FUNCTION_BLOCK RADIO_BOOL (* Radio Button BOOL Input *)
  (* Standard: 61499-1; Classification: HMI *)
  (* Version 0.3, 2004-06-21, JHC, Rockwell Automation, Updated documentation (REQ not inhibited). *)
  (* Version 0.2, 2004-06-08, JHC, Rockwell Automation, Updated documentation (REQ not inhibited). *)
  (* Version 0.1, 2002-05-03, JHC, Rockwell Automation, Made QI IV=true. *)
  (* Version 0.0, 2001-03-03, JHC, Rockwell Automation *)
  (* Compiler header: package fb.rt.hmi; import java.awt.*; import java.awt.event.*; *)
  (* Compiler classdef: public class RADIO_BOOL extends FBInstance implements ItemListener *)
  (* Compiler Java Sun JDK 1.4.2 *)
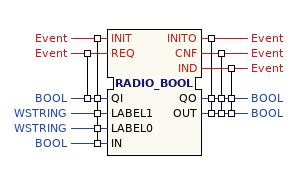
  EVENT_INPUT
    INIT WITH QI, LABEL1, LABEL0, IN; (* Initialization *)
    REQ WITH QI; (* Request *)
  END_EVENT
  EVENT_OUTPUT
    INITO WITH QO, OUT; (* Initialization Confirm *)
    CNF WITH QO, OUT; (* Service Confirmation *)
    IND WITH QO, OUT; (* User changed state *)
  END_EVENT
  VAR_INPUT
    QI : BOOL := true; (* Event qualifier *)
    LABEL1 : WSTRING := TRUE; (* Label for TRUE state *)
    LABEL0 : WSTRING := FALSE; (* Label for FALSE state *)
    IN : BOOL; (* Initial value *)
  END_VAR
  VAR_OUTPUT
    QO : BOOL; (* Event qualifier *)
    OUT : BOOL; (* Output data *)
  END_VAR
  SERVICE RADIO_BOOL/HMI
    SEQUENCE normal_initialization
      RADIO_BOOL.INIT+(LABEL1,LABEL0,IN) -> HMI.initialize() -> RADIO_BOOL.INITO+(OUT);
    END_SEQUENCE
    SEQUENCE initialization_inhibited
      RADIO_BOOL.INIT-() -> RADIO_BOOL.INITO-();
    END_SEQUENCE
    SEQUENCE indication
      HMI.itemStateChanged(QI=1) -> RADIO_BOOL.IND+(OUT);
    END_SEQUENCE
    SEQUENCE indication_inhibited
      HMI.itemStateChanged(QI=0);
    END_SEQUENCE
    SEQUENCE request_no_change
      RADIO_BOOL.REQ+(IN) -> HMI.select() -> RADIO_BOOL.CNF+(OUT);
    END_SEQUENCE
    SEQUENCE request_selection_change
      RADIO_BOOL.REQ+(IN) -> HMI.select() -> RADIO_BOOL.IND+(OUT) -> RADIO_BOOL.CNF+(OUT);
    END_SEQUENCE
    SEQUENCE request_inhibited
      RADIO_BOOL.REQ-() -> RADIO_BOOL.CNF-();
    END_SEQUENCE
  END_SERVICE
END_FUNCTION_BLOCK
